Staubli VAL3: StaubliUI.pjx

--- StaubliUI.pjx ---
Parameters version=s7.3.1 stackSize=15000 millimeterUnit=true
Program file=Bool_Edit.pgx
Program file=BoolMess_Edit.pgx
Program file=Control_Action.pgx
Program file=Control_BatPrt.pgx
Program file=Control_BatSpd.pgx
Program file=Control_Bottom.pgx
Program file=Control_BottomS.pgx
Program file=Control_Joint.pgx
Program file=Control_Lable.pgx
Program file=Control_Left.pgx
Program file=Control_LeftS.pgx
Program file=Control_List.pgx
Program file=Control_List1S.pgx
Program file=Control_ListBS.pgx
Program file=Control_ListCls.pgx
Program file=Control_ListMC.pgx
Program file=Control_ListMCD.pgx
Program file=Control_ListMJ.pgx
Program file=Control_ListS.pgx
Program file=Control_Loffset.pgx
Program file=Control_MCShow.pgx
Program file=Control_Mess.pgx
Program file=Control_Panel.pgx
Program file=Control_PanelB.pgx
Program file=Control_PanelD.pgx
Program file=Control_PanelMd.pgx
Program file=Control_PanelS.pgx
Program file=Control_PanelXY.pgx
Program file=Control_Para.pgx
Program file=Control_PatMove.pgx
Program file=Control_Point.pgx
Program file=Control_Preset.pgx
Program file=Control_Recipe.pgx
Program file=Control_Remote.pgx
Program file=Control_Scara.pgx
Program file=Control_Timer.pgx
Program file=Control_Traj.pgx
Program file=Control_YesNO.pgx
Program file=Float_Edit.pgx
Program file=Form_4jHome.pgx
Program file=Form_6jHome.pgx
Program file=Form_Action.pgx
Program file=Form_Bye.pgx
Program file=Form_Config.pgx
Program file=Form_LabelList.pgx
Program file=Form_Main.pgx
Program file=Form_MainS.pgx
Program file=Form_Panel.pgx
Program file=Form_Panel4P.pgx
Program file=Form_PanelBool.pgx
Program file=Form_PanelJoint.pgx
Program file=Form_PanelList.pgx
Program file=Form_PanelPoint.pgx
Program file=Form_PanelStr.pgx
Program file=Form_Patten.pgx
Program file=Form_PattenD.pgx
Program file=Form_PattenS.pgx
Program file=Form_Product.pgx
Program file=Form_ScaraRobot.pgx
Program file=Form_SelSharp.pgx
Program file=Form_Simulation.pgx
Program file=Form_Welcome.pgx
Program file=Int_Edit.pgx
Program file=Int_EditS.pgx
Program file=Key_ListBase.pgx
Program file=Key_ListMC.pgx
Program file=ReadMe.pgx
Program file=Sel_Edit.pgx
Program file=start.pgx
Program file=stop.pgx
Program file=Str_Edit.pgx
Program file=Str_SplitChar.pgx
Program file=Str_SplitComma.pgx
Data file=StaubliUI.dtx

--- start.pgx ---
public program start()
  local num l_nKeyValue
  local bool l_bBool[199]
  local num l_nNum
  local num l_nNum1
  local bool l_brES
begin
  cls()
  //call Control_PanelB("fasdfa","fasdfas")
//  call Frame_PattenD("hELLO")
//  call Control_ListS("1,3,5,6,6,7,8,8,9,90,2,43,5,56",l_nNum)
//  //call Control_YesNO("FDSAFA  AFSDASA",l_brES)
// // call Control_Timer("fasdfafa",5)
////  cls()
////  if l_brES
////    popUpMsg("yes")
////  else
////    popUpMsg("NO")
////  endIf
//   l_bBool[120]=true
//   call Control_ListMC(l_bBool,l_nNum,l_nNum1)
//   call Control_Lable("目前点序号:",l_nNum,0)
//   while true
//
//    call Key_ListMC(l_brES,l_nKeyValue,l_nNum,l_nNum1)
//    if l_brES
//      call Control_ListMC(l_bBool,l_nNum,l_nNum1)
//      call Control_Lable("目前点序号:",l_nNum,0)
//    endIf
//    //使用Q作为快选方式
//    if l_nKeyValue==113
//     call Num_EditS1D(l_nNum,"目前点序号:")
//     call Control_ListMC(l_bBool,l_nNum,l_nNum1)
//     call Control_Lable("目前点序号:",l_nNum,0)
//
//    endIf
//

//
//
//    delay(0)
//  endWhile
//  call Frame_PattenD("hELLO")
   call Control_ListBS("1,2,3,4,5,6","发生大幅，发，发，发，发，发",l_nNum,0)


end

--- Bool_Edit.pgx ---
public program Bool_Edit(bool& x_bRes, num x_nX, num x_nY, num x_nLength)
  local num l_nNum
  local string l_s[2]
begin

  l_s[1]="是"
  l_s[0]="否"


   call BoolMess_Edit(x_bRes,x_nX,x_nY,x_nLength,l_s)

end

--- BoolMess_Edit.pgx ---
public program BoolMess_Edit(bool& x_bRes, num x_nX, num x_nY, num x_nLength, string& x_sMess[])
  local num l_nNum
begin


   l_nNum=sel(x_bRes,1,0)
   call Sel_Edit(l_nNum,x_nX,x_nY,x_sMess)
   x_bRes=(l_nNum==1)

end

--- Control_Action.pgx ---
public program Control_Action(num& x_nAction[] (dimensions=3), num x_nIndex, string& x_sIoName[], bool& x_bDigtal[])
  local string l_sItem[2]
  local num l_nNum
  local num l_nKey
  local num l_nData[24]
  local num l_nSelectIndex
  local bool l_bRes
begin

  //修改点位的 joint

  for l_nNum=0 to 11
    l_nData[l_nNum*2+0]=x_nAction[x_nIndex,l_nNum,0]
    l_nData[l_nNum*2+1]=x_nAction[x_nIndex,l_nNum,1]
  endFor
  l_sItem[0]="关"
  l_sItem[1]="开"

  resize(sBuff,1,24)


  call Control_BottomS("置空,清空,延时,,,,取消,确定")
  call Control_PanelXY(4,0,20,10)
  call Control_Panel("动作值")
  for l_nNum=0 to 11


    sBuff[l_nNum*2+0]=toString("",l_nNum+1)+"名称:"+x_sIoName[l_nData[l_nNum*2+0]]
    if x_bDigtal[l_nData[l_nNum*2]]
      sBuff[l_nNum*2+1]="值 : "+ l_sItem[sel(l_nData[l_nNum*2+1]==0,0,1)]
    else
      sBuff[l_nNum*2+1]="值 : "+toString("",l_nData[l_nNum*2+1])
    endIf

  endFor
  call Control_List(sBuff,l_nSelectIndex)


  //**********************************
  //按键响应
  while true
    l_nKey=getKey()

    switch l_nKey
      //向上
      case 261
        l_nSelectIndex=max(0,l_nSelectIndex-1)
      break

      //向下
      case 266
        l_nSelectIndex=min(l_nSelectIndex+1,23)
      break

      //编辑
      case 270
        if l_nSelectIndex%2==1
          if ! x_bDigtal[l_nData[l_nSelectIndex-1]]
            call Float_Edit(l_nData[l_nSelectIndex],nPanelLTopX+6,l_nSelectIndex+nPanelLTopY+1)
          else
            call Sel_Edit(l_nData[l_nSelectIndex],nPanelLTopX+6,l_nSelectIndex+nPanelLTopY+1,l_sItem)
          endIf

        else
          call Sel_Edit(l_nData[l_nSelectIndex],nPanelLTopX+7,l_nSelectIndex+nPanelLTopY+1,x_sIoName)
        endIf

      break

      case 271
        call Control_YesNO("确定设置为无IO信号吗?",l_bRes)
        if l_bRes

          l_nData[sel(l_nSelectIndex%2==0,l_nSelectIndex,l_nSelectIndex-1)]=0

        endIf

      break


      //全部置空
      case 272
        call Control_YesNO("确定全部清空吗?",l_bRes)
        if l_bRes
          for l_nNum=0 to 23
            l_nData[l_nNum]=0
          endFor


        endIf
      break


      case 273
        call Control_YesNO("确定要设置为延时吗?",l_bRes)
        if l_bRes
          l_nData[sel(l_nSelectIndex%2==0,l_nSelectIndex,l_nSelectIndex-1)]=165

        endIf
      break


      //退出
      case 277
        cls()
        return

      break



      //取消
      case 278
        for l_nNum=0 to 11
          x_nAction[x_nIndex,l_nNum,0]= l_nData[l_nNum*2+0]
          x_nAction[x_nIndex,l_nNum,1]=l_nData[l_nNum*2+1]
        endFor
        return
      break

    endSwitch

    if l_nKey!=-1

      for l_nNum=0 to 11
        sBuff[l_nNum*2+0]=toString("",l_nNum+1)+"名称:"+x_sIoName[l_nData[l_nNum*2+0]]
        if x_bDigtal[l_nData[l_nNum*2]]
          sBuff[l_nNum*2+1]="值 : "+ l_sItem[sel(l_nData[l_nNum*2+1]==0,0,1)]
        else
          sBuff[l_nNum*2+1]="值 : "+toString("",l_nData[l_nNum*2+1])
        endIf

      endFor

      call Control_PanelXY(4,0,20,10)
      call Control_Panel("动作值")
      call Control_List(sBuff,l_nSelectIndex)
      call Control_BottomS("置空,清空,延时,,,,取消,确定")
    endIf


  endWhile





end

--- Control_BatPrt.pgx ---
public program Control_BatPrt(num& x_nFrom, num& x_nTo, num& x_nPreset)
  local string l_sItem[3]
  local num l_nNum
  local num l_nKey
  local num l_nData[6]
  local num l_nSelectIndex
begin

  //修改点位的 joint
  l_nData[0]=x_nFrom
  l_nData[1]=x_nTo
  l_nData[2]=1
  //l_nData[3]=15
  l_sItem[0]="开始    :"+toString("",l_nData[0])
  l_sItem[1]="结束    :"+toString("",l_nData[1])
  l_sItem[2]="工艺    :"+toString("",l_nData[2])
  //  l_sItem[3]="加速度  :"+toString("",l_nData[3])



  call Control_BottomS(",,,,,,取消,确定")
  call Control_PanelXY(8,0,15,4)
  call Control_Panel("批处理工艺")
  call Control_List(l_sItem,l_nSelectIndex)
  while true
    l_nKey=getKey()

    switch l_nKey
      case 261
        l_nSelectIndex=max(0,l_nSelectIndex-1)
      break

      case 266
        l_nSelectIndex=min(l_nSelectIndex+1,2)
      break

      case 278
        x_nFrom=l_nData[0]
        x_nTo=l_nData[1]
        x_nPreset=l_nData[2]
        //   x_nAcc=l_nData[3]
        cls()
        return
      break


      case 277,255

        cls()
        return
      break

      case 270
        call Float_Edit(l_nData[l_nSelectIndex],nPanelLTopX+7,l_nSelectIndex+nPanelLTopY+1)
      break

    endSwitch

    if l_nKey!=-1
      l_nData[2]=min(max(1,l_nData[2]),50)
      l_nData[2]=round(l_nData[2])
      l_sItem[0]="开始    :"+toString("",l_nData[0])
      l_sItem[1]="结束    :"+toString("",l_nData[1])
      l_sItem[2]="工艺    :"+toString("",l_nData[2])
      // l_sItem[3]="加速度  :"+toString("",l_nData[3])
      call Control_List(l_sItem,l_nSelectIndex)

    endIf






  endWhile





end

--- Control_BatSpd.pgx ---
public program Control_BatSpd(num& x_nFrom, num& x_nTo, num& x_nSpeed, num& x_nAcc)
  local string l_sItem[4]
  local num l_nNum
  local num l_nKey
  local num l_nData[6]
  local num l_nSelectIndex
begin

  //修改点位的 joint
  l_nData[0]=x_nFrom
  l_nData[1]=x_nTo
  l_nData[2]=100
  l_nData[3]=15
  l_sItem[0]="开始    :"+toString("",l_nData[0])
  l_sItem[1]="结束    :"+toString("",l_nData[1])
  l_sItem[2]="速度    :"+toString("",l_nData[2])
  l_sItem[3]="加速度  :"+toString("",l_nData[3])



  call Control_BottomS(",,,,,,取消,确定")
  call Control_PanelXY(8,0,15,4)
  call Control_Panel("批处理速度")
  call Control_List(l_sItem,l_nSelectIndex)
  while true
    l_nKey=getKey()

    switch l_nKey
      case 261
        l_nSelectIndex=max(0,l_nSelectIndex-1)
      break

      case 266
        l_nSelectIndex=min(l_nSelectIndex+1,3)
      break

      case 278
        x_nFrom=l_nData[0]
        x_nTo=l_nData[1]
        x_nSpeed=l_nData[2]
        x_nAcc=l_nData[3]
        cls()
        return
      break


      case 277,255

        cls()
        return
      break

      case 270
        call Float_Edit(l_nData[l_nSelectIndex],nPanelLTopX+7,l_nSelectIndex+nPanelLTopY+1)
      break

    endSwitch

    if l_nKey!=-1
  l_sItem[0]="开始    :"+toString("",l_nData[0])
  l_sItem[1]="结束    :"+toString("",l_nData[1])
  l_sItem[2]="速度    :"+toString("",l_nData[2])
  l_sItem[3]="加速度  :"+toString("",l_nData[3])
      call Control_List(l_sItem,l_nSelectIndex)

    endIf






  endWhile





end

--- Control_Bottom.pgx ---
public program Control_Bottom(string& x_sBottomList[])
  local num l_nIndex
  local num l_nNum
begin
  //说明：
  //函数功能：对功能键进行说明
  //


  //参数初始化
  setTextMode(0)
  l_nNum=min(7,size(x_sBottomList)-1)


  for l_nIndex=0 to  l_nNum
    gotoxy(1+l_nIndex*5,13)
    put(left(x_sBottomList[l_nIndex]+"       ",4+len(x_sBottomList[l_nIndex])-getDisplayLen(x_sBottomList[l_nIndex])))
  endFor

  //补全
  if l_nNum<7
    for l_nIndex=l_nNum to 7
      gotoxy(1+l_nIndex*5,13)
      put("  ")
    endFor
  endIf
end

--- Control_BottomS.pgx ---
public program Control_BottomS(string x_sBottomList)
  local string l_sBottomList[8]
  local bool l_bRes
begin

  call Str_SplitComma(l_bRes,x_sBottomList,l_sBottomList)
  if !l_bRes
    return
  endIf

call Control_Bottom(l_sBottomList)

end

--- Control_Joint.pgx ---
public program Control_Joint(jointRx& x_jJ)
  local string l_sItem[6]
  local num l_nNum
  local num l_nKey
  local num l_nData[6]
  local num l_nSelectIndex
begin

  //修改点位的 joint
  l_nData[0]=x_jJ.j1
  l_nData[1]=x_jJ.j2
  l_nData[2]=x_jJ.j3
  l_nData[3]=x_jJ.j4
  l_nData[4]=x_jJ.j5
  l_nData[5]=x_jJ.j6

  for l_nNum=0 to 5
    l_sItem[l_nNum]="j"+toString("",l_nNum+1)+"   :"+toString(".3",l_nData[l_nNum])
  endFor

  call Control_BottomS(",,,,,,取消,确定")
  call Control_PanelXY(8,0,15,6)
  call Control_Panel("Joint值")
  call Control_List(l_sItem,l_nSelectIndex)
  while true
    l_nKey=getKey()

    switch l_nKey
      case 261
        l_nSelectIndex=max(0,l_nSelectIndex-1)
      break

      case 266
        l_nSelectIndex=min(l_nSelectIndex+1,5)
      break

      case 278
        x_jJ.j1=l_nData[0]
        x_jJ.j2=l_nData[1]
        x_jJ.j3=l_nData[2]
        x_jJ.j4=l_nData[3]
        x_jJ.j5=l_nData[4]
        x_jJ.j6=l_nData[5]
        return
      break


      case 277,255
        return
      break

      case 270
        call Float_Edit(l_nData[l_nSelectIndex],nPanelLTopX+7,l_nSelectIndex+nPanelLTopY+1)
      break

    endSwitch

    if l_nKey!=-1
      for l_nNum=0 to 5
        l_sItem[l_nNum]="j"+toString("",l_nNum+1)+"   :"+toString(".3",l_nData[l_nNum])
      endFor
      call Control_List(l_sItem,l_nSelectIndex)

    endIf






  endWhile





end

--- Control_Lable.pgx ---
public program Control_Lable(string x_sMess, num& Value, num x_nTextMode)
begin
setTextMode(0)
gotoxy(0,0)
put(x_sMess)
gotoxy(getDisplayLen(x_sMess),0)
x_nTextMode=min(max(0,x_nTextMode),3)
setTextMode(x_nTextMode)
//序号加1
put(left(toString("",Value+1)+"            ",max(8,nPanelLTopX-getDisplayLen(x_sMess)-len(toString("",Value)))))
setTextMode(0)
end

--- Control_Left.pgx ---
program Control_Left(string& x_sLeftList[])
  local num l_nIndex
begin

    setTextMode(0)
  //左边栏进行显示
  for l_nIndex=0 to min(7,size(x_sLeftList)-1)
    gotoxy(1,l_nIndex+4)
    if size(x_sLeftList)>l_nIndex and x_sLeftList[l_nIndex]!=""
      put("F"+toString("",l_nIndex+1)+"->"+x_sLeftList[l_nIndex])
    endIf
  endFor
end

--- Control_LeftS.pgx ---
public program Control_LeftS(string x_sLeftList)
  local bool l_bRes
  local string l_sBuff[20]
begin

  call Str_SplitComma(l_bRes,x_sLeftList,l_sBuff)
  if !l_bRes
    return
  endIf

call Control_Left(l_sBuff)
end

--- Control_List.pgx ---
public program Control_List(string& x_sItemName[], num& x_nSelectItem)
  local num l_nIndex
  local bool l_bRes
  local num l_nFrist
  local num l_nNum
  local bool l_bBlack
  local bool l_bBlank
  local num l_nCount
begin
  //说明：
  //函数功能：在划定的框内，把选中项给显示出来
  //l_nFirst  在列表中第一个显示的项的序号
  //x_nSelectItem  被选中的项的序号
  //l_nCount 合法列表项的项总数，如何数组中间为空，则可能被截断


  //1.参数初始化
  l_nFrist=0
  l_nCount=0

  //2.参数合法化判断，得到合法项的总数
  for l_nIndex=0 to size(x_sItemName)-1
    if x_sItemName[l_nIndex]==""
      l_nIndex=size(x_sItemName)
    else
      l_nCount=l_nCount+1
    endIf
  endFor

  //3.如果选中项大于列表长度
  x_nSelectItem=min(max(0,x_nSelectItem),l_nCount-1)
  if x_nSelectItem>=nPanelLengthY
    l_nFrist=x_nSelectItem-nPanelLengthY+1
  endIf


  //4.把列表给画出来
  for l_nIndex=0 to min(nPanelLengthY-1,l_nCount-l_nFrist-1)
    gotoxy(nPanelLTopX+1,nPanelLTopY+l_nIndex+1)
    setTextMode(sel(l_nIndex+l_nFrist==x_nSelectItem,1,0))
    l_nNum=nPanelWidthX-getDisplayLen(x_sItemName[l_nIndex+l_nFrist])+len(x_sItemName[l_nIndex+l_nFrist])
    put(left(x_sItemName[l_nIndex+l_nFrist]+"                            ",l_nNum))
  endFor


  //5.对剩下的进行补空
  setTextMode(0)
  while l_nIndex< nPanelLengthY
    gotoxy(nPanelLTopX+1,nPanelLTopY+l_nIndex+1)
    put(left("                               ",nPanelWidthX-2))
    l_nIndex=l_nIndex+1
  endWhile


end

--- Control_List1S.pgx ---
public program Control_List1S(string x_sItemName, string x_sItemValue, num x_nSelectItem, num x_nText)
  local string l_sBuff[10]
  local string l_sValue[10]
  local num l_nIndex
  local bool l_bRes
begin
   // 赋初值
   for l_nIndex=0 to size(l_sBuff)-1
    l_sBuff[l_nIndex]=""
  endFor

  //把项的名字给解析出来
  call  Str_SplitChar(l_bRes,x_sItemName,",",l_sBuff)
  if !l_bRes
    return
  endIf

    call  Str_SplitChar(l_bRes,x_sItemValue,",",l_sValue)
  if !l_bRes
    return
  endIf


  //对方框的定义进行赋初值
  // call Control_ListBas(x_nSelectItem)


  //把列表给画出来
  for l_nIndex=0 to min(min(nPanelLengthY-1,size(l_sBuff)-1),size(l_sValue)-1)
    if l_sBuff[l_nIndex]==""
      return
    endIf
    setTextMode(0)
    gotoxy(nPanelLTopX+1,nPanelLTopX+l_nIndex+1)
    put(left(l_sBuff[l_nIndex]+"              ",nPanelWidthX-getDisplayLen(l_sBuff[l_nIndex])+len(l_sBuff[l_nIndex]))+":")
    gotoxy(nPanelLTopX+nPanelWidthX/2-getDisplayLen(l_sBuff[l_nIndex])+len(l_sBuff[l_nIndex]),nPanelLTopY+l_nIndex+1)
    //选中项变成黑色
    if l_nIndex==x_nSelectItem

      setTextMode(x_nText)
    endIf

    //直接截取+
    //中文编码与英文编码有点不一样
    put(left(l_sValue[l_nIndex]+"             ",nPanelWidthX/2-getDisplayLen(l_sValue[l_nIndex])+len(l_sValue[l_nIndex])))

  endFor


end

--- Control_ListBS.pgx ---
public program Control_ListBS(string x_sItemName, string x_sItemValue, num x_nSelectItem, num x_nText)
  local string l_sBuff[10]
  local string l_sValue[10]
  local num l_nIndex
  local bool l_bRes
begin
   // 赋初值
   for l_nIndex=0 to size(l_sBuff)-1
    l_sBuff[l_nIndex]=""
  endFor

  //把项的名字给解析出来
  call  Str_SplitComma(l_bRes,x_sItemName,l_sBuff)
  if !l_bRes
    return
  endIf

    call  Str_SplitComma(l_bRes,x_sItemValue,l_sValue)
  if !l_bRes
    return
  endIf

  call Control_PanelXY(nPanelLTopX,nPanelLTopY,nPanelWidthX/2,nPanelLengthY)
  call Control_List(l_sBuff,x_nSelectItem)
  call Control_PanelXY(nPanelLTopX+nPanelWidthX/2,nPanelLTopY,nPanelWidthX/2,nPanelLengthY)
  call Control_List(l_sValue,x_nSelectItem)

end

--- Control_ListCls.pgx ---
program Control_ListCls()
  local num l_nIndex
begin



  //对方框的定义进行赋初值
  if nPanelLengthY<=0 and nPanelLTopX<=0 and nPanelLTopY<=0 and nPanelWidthX<=0
    call Control_PanelXY(20,0,18,11)
  endIf

  //清空列表
  setTextMode(0)
  for l_nIndex=0 to nPanelLengthY-1
    gotoxy(nPanelLTopX+1,nPanelLTopY+l_nIndex+1)
    put(left("                                               ",nPanelWidthX))
  endFor

  //参数判断  对于选择项的判断
 // x_nSelectItem=min(max(0,x_nSelectItem),nPanelLengthY-1)


end

--- Control_ListMC.pgx ---
public program Control_ListMC(bool& x_bMC[], num& x_nSelectItem, num x_nText)
  local num l_nIndex
  local bool l_bRes
  local string l_sText
  local num l_nFrist
begin
   //赋初值
   // call Control_ListCls()

    l_nFrist=0
  x_nSelectItem=min(max(0,x_nSelectItem),size(x_bMC)-1)
  if x_nSelectItem>=nPanelLengthY
    l_nFrist=x_nSelectItem-nPanelLengthY+1
  endIf


  //把列表给画出来
  for l_nIndex=0 to min(nPanelLengthY-1,size(x_bMC)-l_nFrist)
    gotoxy(nPanelLTopX+1,nPanelLTopY+l_nIndex+1)
    //选中项变成黑色


    //MOVEL
    if !x_bMC[l_nIndex+l_nFrist]
      if l_nIndex+l_nFrist==x_nSelectItem

        setTextMode(1)
      else
        setTextMode(0)
      endIf
      put(left(toString("",l_nIndex+l_nFrist+1)+"       ",5 )+left("MOVEL             ",nPanelWidthX-5))
    else

    //MOVEC
       setTextMode(0)
      put(left("                                               ",nPanelWidthX))
      gotoxy(nPanelLTopX+1,nPanelLTopY+l_nIndex+1)
      if l_nIndex+l_nFrist!=x_nSelectItem
        put(left(toString("",l_nIndex+l_nFrist+1)+"       ",5 )+left("MOVEC Pc Pt              ",nPanelWidthX-5))
      else
        if x_nText==0
          setTextMode(1)
        else
          setTextMode(0)
        endIf
        put(left(toString("",l_nIndex+l_nFrist+1)+"       ",5 )+"MOVEC")
        gotoxy(nPanelLTopX+12,nPanelLTopY+l_nIndex+1)
        if x_nText==1

          setTextMode(1)
        else
          setTextMode(0)
        endIf
        put("Pc")
        //目标点
        gotoxy(nPanelLTopX+15,nPanelLTopY+l_nIndex+1)

        if x_nText==2
          setTextMode(1)
        else
          setTextMode(0)
        endIf
        put("Pt")
      endIf
    endIf
  endFor

   setTextMode(0)
  while l_nIndex< nPanelLengthY
    gotoxy(nPanelLTopX+1,nPanelLTopY+l_nIndex+1)
    put(left("                          ",nPanelWidthX-2))
    l_nIndex=l_nIndex+1
  endWhile

end

--- Control_ListMCD.pgx ---
public program Control_ListMCD(bool& x_bMC[], num& x_nSelectItem, num& x_nText)
  local num l_nIndex
  local bool l_bRes
  local string l_sText
  local num l_nFrist
begin
   //赋初值
   // call Control_ListCls()

    l_nFrist=0
  x_nSelectItem=min(max(0,x_nSelectItem),size(x_bMC)-1)
  if x_nSelectItem>=nPanelLengthY
    l_nFrist=x_nSelectItem-nPanelLengthY+1
  endIf


  //把列表给画出来
  for l_nIndex=0 to min(nPanelLengthY-1,size(x_bMC)-l_nFrist)
    gotoxy(nPanelLTopX+1,nPanelLTopY+l_nIndex+1)
    //选中项变成黑色


    //MOVEL
    if !x_bMC[l_nIndex+l_nFrist]
      if l_nIndex+l_nFrist==x_nSelectItem
          if x_nText==0
          setTextMode(1)
        else
          setTextMode(0)
        endIf
        put(left(toString("",l_nIndex+l_nFrist+1)+"       ",5 )+"MOVEL")
        gotoxy(nPanelLTopX+12,nPanelLTopY+l_nIndex+1)
        if x_nText==1

          setTextMode(1)
        else
          setTextMode(0)
        endIf
        put("Pl")
      else
        setTextMode(0)
        put(left(toString("",l_nIndex+l_nFrist+1)+"       ",5 )+left("MOVEL Pl             ",nPanelWidthX-5))
      endIf

    else

    //MOVEC
       setTextMode(0)
      put(left("                                               ",nPanelWidthX))
      gotoxy(nPanelLTopX+1,nPanelLTopY+l_nIndex+1)
      if l_nIndex+l_nFrist!=x_nSelectItem
        put(left(toString("",l_nIndex+l_nFrist+1)+"       ",5 )+left("MOVEC Pc Pt              ",nPanelWidthX-5))
      else
        if x_nText==0
          setTextMode(1)
        else
          setTextMode(0)
        endIf
        put(left(toString("",l_nIndex+l_nFrist+1)+"       ",5 )+"MOVEC")
        gotoxy(nPanelLTopX+12,nPanelLTopY+l_nIndex+1)
        if x_nText==1

          setTextMode(1)
        else
          setTextMode(0)
        endIf
        put("Pc")
        //目标点
        gotoxy(nPanelLTopX+15,nPanelLTopY+l_nIndex+1)

        if x_nText==2
          setTextMode(1)
        else
          setTextMode(0)
        endIf
        put("Pt")
      endIf
    endIf
  endFor

   setTextMode(0)
  while l_nIndex< nPanelLengthY
    gotoxy(nPanelLTopX+1,nPanelLTopY+l_nIndex+1)
    put(left("                          ",nPanelWidthX-2))
    l_nIndex=l_nIndex+1
  endWhile

end

--- Control_ListMJ.pgx ---
public program Control_ListMJ(bool& x_bMJ[], num x_nMoveFirst, num x_nSelectItem)
  local num l_nIndex
  local bool l_bRes
  local string l_sText
begin


//  call Control_ListBas(x_nSelectItem)
//
//
//
//
//  //把列表给画出来
//  for l_nIndex=0 to min(nBottomY-nTopY-1,size(x_bMJ)-x_nMoveFirst)
//
//    setTextMode(0)
//    if x_nMoveFirst+l_nIndex>size(x_bMJ)-1
//      return
//    endIf
//    //MOVEL
//    gotoxy(nTopX+1,nTopY+l_nIndex+1)
//    if !x_bMJ[x_nMoveFirst+l_nIndex]
//      if l_nIndex==x_nSelectItem
//        setTextMode(1)
//      else
//        setTextMode(0)
//      endIf
//      put(left(toString("",x_nMoveFirst+l_nIndex+1)+"       ",4 )+left("MOVEJ             ",24-nBottomX))
//    else
//      //MOVEC
//      if l_nIndex==x_nSelectItem
//        setTextMode(1)
//      else
//        setTextMode(0)
//      endIf
//      put(left(toString("",x_nMoveFirst+l_nIndex+1)+"       ",4 )+left("MOVEL              ",24-nBottomX))
//
//    endIf
//
//  endFor
//

end

--- Control_ListS.pgx ---
program Control_ListS(string x_sItemName, num& x_nSelectItem)
  local bool l_bRes
  local string l_sBuff[20]
begin

 call Str_SplitComma(l_bRes,x_sItemName,l_sBuff)
 if !l_bRes
  return
endIf
  call Control_List(l_sBuff,x_nSelectItem)


end

--- Control_Loffset.pgx ---
public program Control_Loffset(num& x_nFrom, num& x_nTo)
  local string l_sItem[2]
  local num l_nNum
  local num l_nKey
  local num l_nData[6]
  local num l_nSelectIndex
begin

  //修改点位的 joint
l_nData[0]=x_nFrom
l_nData[1]=x_nTo

  l_sItem[0]="开始    :"+toString("",l_nData[0])
  l_sItem[1]="停止    :"+toString("",l_nData[1])
  call Control_BottomS(",,,,,,取消,确定")
  call Control_PanelXY(8,0,15,6)
  call Control_Panel("局部偏差值")
  call Control_List(l_sItem,l_nSelectIndex)
  while true
    l_nKey=getKey()

    switch l_nKey
      case 261
        l_nSelectIndex=max(0,l_nSelectIndex-1)
      break

      case 266
        l_nSelectIndex=min(l_nSelectIndex+1,1)
      break

      case 278
          x_nFrom=l_nData[0]
          x_nTo=l_nData[1]
         cls()
        return
      break


      case 277,255

        cls()
        return
      break

      case 270
        call Float_Edit(l_nData[l_nSelectIndex],nPanelLTopX+7,l_nSelectIndex+nPanelLTopY+1)
      break

    endSwitch

    if l_nKey!=-1
  l_sItem[0]="开始    :"+toString("",l_nData[0])
  l_sItem[1]="停止    :"+toString("",l_nData[1])
      call Control_List(l_sItem,l_nSelectIndex)

    endIf






  endWhile





end

--- Control_MCShow.pgx ---
public program Control_MCShow(num x_nIndex, num x_nMoveType)
  local string l_sS[3]
begin
  if x_nMoveType>2 or x_nMoveType<1
    return
  endIf
  l_sS[0]=toString("",x_nIndex+1)+"."+"MoveC "
  l_sS[1]=toString("",1)+" "
  l_sS[2]=left(" "+toString("",2)+"       ",nPanelWidthX-len(l_sS[0])-len(l_sS[1]))
  setTextMode(0)
  gotoxy(nPanelLTopX+1,min(nPanelLengthY,x_nIndex+1))
  put(l_sS[0])
  setTextMode(sel(x_nMoveType==1,1,0))
  put(l_sS[1])
  setTextMode(sel(x_nMoveType==1,0,1))
  put(l_sS[2])


  setTextMode(0)

end

--- Control_Mess.pgx ---
public program Control_Mess(string x_sMess, string x_sLable)
begin

  setTextMode(0)
gotoxy(0,1)
put(x_sMess)
  gotoxy(0,2)
put(x_sLable)

end

--- Control_Panel.pgx ---
program Control_Panel(string x_sTitle)
  local num l_nIndex
  local string l_sS
begin
  //画框函数
  //如果标题为空，



    setTextMode(0)

  //方框进行重画

  //画上边
   gotoxy(nPanelLTopX,nPanelLTopY)
   l_sS="┌"+left("───────────────────────────────────",nPanelWidthX)

  //写标题

     //2是两个标志符
  if x_sTitle!=""
    x_sTitle=left(x_sTitle,min(getDisplayLen(x_sTitle),nPanelWidthX)-getDisplayLen(x_sTitle)+len(x_sTitle))
    x_sTitle="┤"+x_sTitle+"├┐"
    l_sS=left(l_sS,nPanelWidthX-getDisplayLen(x_sTitle)+2)+x_sTitle
  else
    l_sS=l_sS+"┐"
  endIf
  put(l_sS)

   //画下边
   gotoxy(nPanelLTopX,nPanelLTopY+nPanelLengthY+1)
   put("└"+left("─────────────────────────────────────────",nPanelWidthX)+"┘")

   //重画两边
   for l_nIndex=1 to nPanelLengthY
    gotoxy(nPanelLTopX,nPanelLTopY+l_nIndex)
   // put("│")
   put("│")
    gotoxy(nPanelLTopX+nPanelWidthX+1,nPanelLTopY+l_nIndex)
    put("│")
  endFor












end

--- Control_PanelB.pgx ---
public program Control_PanelB(string x_sLeftTitle, string x_sRightTitle)
begin
    //两个方框
   call Control_PanelS(x_sLeftTitle,0,0,18,11)

   call Control_PanelS(x_sRightTitle,20,0,18,11)

end

--- Control_PanelD.pgx ---
public program Control_PanelD()
begin
  call Control_PanelS("",20,0,18,11)


end

--- Control_PanelMd.pgx ---
public program Control_PanelMd(string x_sMess)
begin

  call Control_PanelS("",2,3,34,4)
  call Control_ListCls()
  x_sMess=left(x_sMess,min(getDisplayLen(x_sMess),nPanelWidthX))
  gotoxy(nPanelLTopX+ (nPanelWidthX-getDisplayLen(x_sMess))/2,nPanelLTopY+nPanelLengthY/2+1)
  put( x_sMess)


end

--- Control_PanelS.pgx ---
public program Control_PanelS(string x_sTitle, num x_nLTopX, num x_nLTopY, num x_nWidthX, num x_nLengthY)
  local num l_nIndex
begin
  //画有标题的框



  //设定框的位置与大小
  call Control_PanelXY(x_nLTopX,x_nLTopY,x_nWidthX,x_nLengthY)

  //文本显示状况进行设定
   call Control_Panel(x_sTitle)









end

--- Control_PanelXY.pgx ---
public program Control_PanelXY(num x_nPanelLTopX, num x_nPanelLTopY, num x_nPanelWidthX, num x_nPanelLengthY)
begin

//对于新建的框和列表进行位置和大小的设定

//对于数值范围进行判断，一般的情况可以使用min,max就可以
//如果传入的参数不正确，则设定初始值
nPanelLTopX=min(max(0,x_nPanelLTopX),38)
nPanelLTopY=min(max(0,x_nPanelLTopY),12)

nPanelWidthX=min(max(0,x_nPanelWidthX),38)
nPanelLengthY=min(max(0,x_nPanelLengthY),12)


end

--- Control_Para.pgx ---
public program Control_Para(trsf& x_trTrsf, bool& x_bRes, bool x_bCut, num x_nType)
  local string l_sItem[6]
  local num l_nNum
  local num l_nKey
  local num l_nData[6]
  local num l_nSelectIndex
begin

  //修改点位的 joint
  l_nData[3]=x_trTrsf.x
  l_nData[4]=x_trTrsf.y
  l_nData[0]=x_trTrsf.z
  l_nData[1]=x_trTrsf.rx

  l_nData[2]=x_trTrsf.ry
  l_nData[5]=x_trTrsf.rz
  l_nNum=sel(x_bRes,1,0)
  resize(sData,1,2)
  if x_bCut

    sData[0]="直线"
    sData[1]="圆弧"
    l_sItem[0]="速度(mm/s:"+toString(".3",l_nData[0])
    l_sItem[1]="加速度(%):"+toString(".3",l_nData[1])
    l_sItem[2]="BLend(mm):"+toString(".3",l_nData[2])
    l_sItem[3]="工艺     :"+toString(".3",l_nData[3])
    l_sItem[4]="动作     :"+toString(".3",l_nData[4])
    l_sItem[5]="圆弧/直线:"+sData[l_nNum]

  else
    sData[0]="MoveJ"
    sData[1]="MoveL"
    l_sItem[0]="速度(mm/s:"+toString(".3",l_nData[0])
    l_sItem[1]="加速度(%):"+toString(".3",l_nData[1])
    l_sItem[2]="关节/直线:"+sData[l_nNum]

  endIf

  call Control_BottomS(",,,,,,取消,确定")
  if x_bCut
    if x_nType!=10
      call Control_PanelXY(8,0,18,5)
    else
      call Control_PanelXY(8,0,18,6)
    endIf
  else
    call Control_PanelXY(8,0,17,3)
  endIf
  call Control_Panel("参数")
  call Control_List(l_sItem,l_nSelectIndex)
  while true
    l_nKey=getKey()

    switch l_nKey
      case 261
        l_nSelectIndex=max(0,l_nSelectIndex-1)
      break

      case 266
        if x_bCut
          if x_nType==10
            l_nSelectIndex=min(l_nSelectIndex+1,5)
          else
            l_nSelectIndex=min(l_nSelectIndex+1,4)
          endIf
        else
          l_nSelectIndex=min(l_nSelectIndex+1,2)
        endIf
      break

      case 278
        x_trTrsf.x=l_nData[3]
        x_trTrsf.y=l_nData[4]
        x_trTrsf.z=l_nData[0]
        x_trTrsf.rx=l_nData[1]

        x_trTrsf.ry=l_nData[2]
        x_trTrsf.rz=l_nData[5]
        x_bRes=(l_nNum==1)
        cls()
        return
      break


      case 277,255
        cls()
        return
      break



      case 270
        if (l_nSelectIndex==2 and !x_bCut) or (l_nSelectIndex==5 and x_bCut)
          call Sel_Edit(l_nNum,nPanelLTopX+11,l_nSelectIndex+nPanelLTopY+1,sData)

        else
          call Float_Edit(l_nData[l_nSelectIndex],nPanelLTopX+11,l_nSelectIndex+nPanelLTopY+1)
        endIf
      break

    endSwitch

    if l_nKey!=-1
      if x_bCut

        sData[0]="直线"
        sData[1]="圆弧"
        l_sItem[0]="速度(mm/s:"+toString(".3",l_nData[0])
        l_sItem[1]="加速度(%):"+toString(".3",l_nData[1])
        l_sItem[2]="BLend(mm):"+toString(".3",l_nData[2])
        l_sItem[3]="工艺     :"+toString(".3",l_nData[3])
        l_sItem[4]="动作     :"+toString(".3",l_nData[4])
        l_sItem[5]="圆弧/直线:"+sData[l_nNum]

      else
        sData[0]="MoveJ"
        sData[1]="MoveL"
        l_sItem[0]="速度(mm/s:"+toString(".3",l_nData[0])
        l_sItem[1]="加速度(%):"+toString(".3",l_nData[1])
        l_sItem[2]="关节/直线:"+sData[l_nNum]

      endIf
      call Control_List(l_sItem,l_nSelectIndex)

    endIf






  endWhile





end

--- Control_PatMove.pgx ---
public program Control_PatMove(num& x_nStart, num& x_nEnd)
  local string l_sItem[6]
  local num l_nNum
  local num l_nKey
  local num l_nData[6]
  local num l_nSelectIndex
begin

  //修改点位的 joint
  l_nData[0]=x_nStart
  l_nData[1]=x_nEnd


  l_sItem[0]="开始模拟点:"+toString(".3",l_nData[0])
  l_sItem[1]="结束模拟点:"+toString(".3",l_nData[1])


  call Control_BottomS(",,,,,,,确定")
  call Control_PanelXY(8,0,15,2)
  call Control_Panel("切割点局部模拟")
  call Control_List(l_sItem,l_nSelectIndex)
  while true
    l_nKey=getKey()

    switch l_nKey
      case 261
        l_nSelectIndex=max(0,l_nSelectIndex-1)
      break

      case 266
        l_nSelectIndex=min(l_nSelectIndex+1,1)
      break

      case 278
        x_nStart=l_nData[0]
        x_nEnd=l_nData[1]
         cls()
        return
      break


//      case 277,255
//
//        cls()
//        return
//      break

      case 270
        call Float_Edit(l_nData[l_nSelectIndex],nPanelLTopX+12,l_nSelectIndex+nPanelLTopY+1)
      break

    endSwitch

    if l_nKey!=-1
  l_sItem[0]="开始模拟点:"+toString(".3",l_nData[0])
  l_sItem[1]="结束模拟点:"+toString(".3",l_nData[1])

      call Control_List(l_sItem,l_nSelectIndex)

    endIf






  endWhile





end

--- Control_Point.pgx ---
public program Control_Point(pointRx& x_pP)
  local string l_sItem[6]
  local num l_nNum
  local num l_nKey
  local num l_nData[6]
  local num l_nSelectIndex
begin

  //修改点位的 joint
  l_nData[0]=x_pP.trsf.x
  l_nData[1]=x_pP.trsf.y
  l_nData[2]=x_pP.trsf.z
  l_nData[3]=x_pP.trsf.rx
  l_nData[4]=x_pP.trsf.ry
  l_nData[5]=x_pP.trsf.rz

  l_sItem[0]="X    :"+toString(".3",l_nData[0])
  l_sItem[1]="y    :"+toString(".3",l_nData[1])
  l_sItem[2]="Z    :"+toString(".3",l_nData[2])
  l_sItem[3]="RX   :"+toString(".3",l_nData[3])
  l_sItem[4]="RY   :"+toString(".3",l_nData[4])
  l_sItem[5]="RZ   :"+toString(".3",l_nData[5])

  call Control_BottomS(",,,,,,取消,确定")
  call Control_PanelXY(8,0,15,6)
  call Control_Panel("Point值")
  call Control_List(l_sItem,l_nSelectIndex)
  while true
    l_nKey=getKey()

    switch l_nKey
      case 261
        l_nSelectIndex=max(0,l_nSelectIndex-1)
      break

      case 266
        l_nSelectIndex=min(l_nSelectIndex+1,5)
      break

      case 278
        x_pP.trsf.x=l_nData[0]
        x_pP.trsf.y=l_nData[1]
        x_pP.trsf.z=l_nData[2]
        x_pP.trsf.rx=l_nData[3]
        x_pP.trsf.ry=l_nData[4]
        x_pP.trsf.rz=l_nData[5]
         cls()
        return
      break


      case 277,255

        cls()
        return
      break

      case 270
        call Float_Edit(l_nData[l_nSelectIndex],nPanelLTopX+7,l_nSelectIndex+nPanelLTopY+1)
      break

    endSwitch

    if l_nKey!=-1
      l_sItem[0]="X    :"+toString(".3",l_nData[0])
      l_sItem[1]="y    :"+toString(".3",l_nData[1])
      l_sItem[2]="Z    :"+toString(".3",l_nData[2])
      l_sItem[3]="RX   :"+toString(".3",l_nData[3])
      l_sItem[4]="RY   :"+toString(".3",l_nData[4])
      l_sItem[5]="RZ   :"+toString(".3",l_nData[5])
      call Control_List(l_sItem,l_nSelectIndex)

    endIf






  endWhile





end

--- Control_Preset.pgx ---
public program Control_Preset(num& x_nPreset[] (dimensions=2), num x_nIndex)
  local string l_sItem[5]
  local num l_nNum
  local num l_nKey
  local num l_nData[5]
  local num l_nSelectIndex
begin

  //修改点位的 joint

  for l_nNum=0 to 4
    l_nData[l_nNum]=x_nPreset[x_nIndex,l_nNum]
  endFor



  l_sItem[0]="激光功率  :"+toString("",l_nData[0])
  l_sItem[1]="气体压力  :"+toString("",l_nData[1])
  l_sItem[2]="占空比频率:"+toString("",l_nData[2])
  l_sItem[3]="激光占空比:"+toString("",l_nData[3])
  l_sItem[4]="随动高度  :"+toString("",l_nData[4])

  call Control_BottomS(",,,,,,取消,确定")
  call Control_PanelXY(8,0,15,5)
  call Control_Panel("工艺值")
  call Control_List(l_sItem,l_nSelectIndex)
  while true
    l_nKey=getKey()

    switch l_nKey
      case 261
        l_nSelectIndex=max(0,l_nSelectIndex-1)
      break

      case 266
        l_nSelectIndex=min(l_nSelectIndex+1,5)
      break

      case 278
        for l_nNum=0 to 4
          x_nPreset[x_nIndex,l_nNum]=min(max(l_nData[l_nNum],0),100)
        endFor
        return
      break


      case 277
        return
      break

      case 270
        call Float_Edit(l_nData[l_nSelectIndex],nPanelLTopX+12,l_nSelectIndex+nPanelLTopY+1)
        l_nData[l_nSelectIndex]=min(max(l_nData[l_nSelectIndex],0),100)
      break

    endSwitch

    if l_nKey!=-1

      l_sItem[0]="激光功率  :"+toString("",l_nData[0])
      l_sItem[1]="气体压力  :"+toString("",l_nData[1])
      l_sItem[2]="占空比频率:"+toString("",l_nData[2])
      l_sItem[3]="激光占空比:"+toString("",l_nData[3])
      l_sItem[4]="随动高度  :"+toString("",l_nData[4])
      call Control_List(l_sItem,l_nSelectIndex)

    endIf






  endWhile





end

--- Control_Recipe.pgx ---
public program Control_Recipe(trsf& x_trFrame, trsf& x_trOffset)
  local num l_nSelectIndex
  local num l_nData[30]
  local num l_nKey
  local num l_nNum
begin
//产品的参数



  //主要是用户坐标系和偏移
  l_nData[0]=x_trFrame.x
  l_nData[1]=x_trFrame.y
  l_nData[2]=x_trFrame.z
  l_nData[3]=x_trFrame.rx
  l_nData[4]=x_trFrame.ry
  l_nData[5]=x_trFrame.rz

  l_nData[6]=x_trOffset.x
  l_nData[7]=x_trOffset.y
  l_nData[8]=x_trOffset.z
  l_nData[9]=x_trOffset.rx
  l_nData[10]=x_trOffset.ry
  l_nData[11]=x_trOffset.rz


  resize(sBuff,1,12)

  sBuff[0]="坐标系X  :"+toString(".3",l_nData[0])
  sBuff[1]="坐标系y  :"+toString(".3",l_nData[1])
  sBuff[2]="坐标系Z  :"+toString(".3",l_nData[2])
  sBuff[3]="坐标系RX :"+toString(".3",l_nData[3])
  sBuff[4]="坐标系RY :"+toString(".3",l_nData[4])
  sBuff[5]="坐标系RZ :"+toString(".3",l_nData[5])


  sBuff[6]="偏移 X   :"+toString(".3",l_nData[6])
  sBuff[7]="偏移 y   :"+toString(".3",l_nData[7])
  sBuff[8]="偏移 Z   :"+toString(".3",l_nData[8])
  sBuff[9]="偏移 RX  :"+toString(".3",l_nData[9])
  sBuff[10]="偏移 RY  :"+toString(".3",l_nData[10])
  sBuff[11]="偏移 RZ  :"+toString(".3",l_nData[11])





  call Control_BottomS(",,,,,,取消,确定")
  call Control_PanelXY(8,0,17,12)
  call Control_Panel("产品参数")
  call Control_List(sBuff,l_nSelectIndex)
  while true
    l_nKey=getKey()

    switch l_nKey
      case 261
        //        l_nSelectIndex=max(0,l_nSelectIndex-1)

        l_nSelectIndex=l_nSelectIndex-1
        if l_nSelectIndex<=-1
          l_nSelectIndex=size(sBuff)-1
        endIf

      break

      case 266
        l_nSelectIndex=l_nSelectIndex+1
        if l_nSelectIndex>=size(sBuff)
          l_nSelectIndex=0
        endIf
        //l_nSelectIndex=min(l_nSelectIndex+1,size(sBuff)-1)
      break

      case 278
        x_trFrame.x=l_nData[0]
        x_trFrame.y =l_nData[1]
        x_trFrame.z=l_nData[2]
        x_trFrame.rx =l_nData[3]
        x_trFrame.ry =l_nData[4]
        x_trFrame.rz =l_nData[5]

        x_trOffset.x=l_nData[6]
        x_trOffset.y =l_nData[7]
        x_trOffset.z =l_nData[8]
        x_trOffset.rx =l_nData[9]
        x_trOffset.ry =l_nData[10]
        x_trOffset.rz =l_nData[11]




        cls()
        return
      break


      case 277
        cls()
        return
      break

      case 270
        call Float_Edit(l_nData[l_nSelectIndex],nPanelLTopX+11,l_nSelectIndex+nPanelLTopY+1)

      break


    endSwitch

    if l_nKey!=-1

      sBuff[0]="坐标系X  :"+toString(".3",l_nData[0])
      sBuff[1]="坐标系y  :"+toString(".3",l_nData[1])
      sBuff[2]="坐标系Z  :"+toString(".3",l_nData[2])
      sBuff[3]="坐标系RX :"+toString(".3",l_nData[3])
      sBuff[4]="坐标系RY :"+toString(".3",l_nData[4])
      sBuff[5]="坐标系RZ :"+toString(".3",l_nData[5])


      sBuff[6]="偏移 X   :"+toString(".3",l_nData[6])
      sBuff[7]="偏移 y   :"+toString(".3",l_nData[7])
      sBuff[8]="偏移 Z   :"+toString(".3",l_nData[8])
      sBuff[9]="偏移 RX  :"+toString(".3",l_nData[9])
      sBuff[10]="偏移 RY  :"+toString(".3",l_nData[10])
      sBuff[11]="偏移 RZ  :"+toString(".3",l_nData[11])
      call Control_List(sBuff,l_nSelectIndex)

    endIf


  endWhile



end

--- Control_Remote.pgx ---
public program Control_Remote(num& x_nMode, num& x_nCycleCount)
  local string l_sItem[2]
  local num l_nNum
  local num l_nKey
  local num l_nData[2]
  local num l_nSelectIndex
  local string l_sSMess[6]
begin

  //修改点位的 joint
  l_nData[0]=max(round(x_nMode),0)
  l_nData[1]=max(round(x_nCycleCount),0)

  l_sSMess[0]="按钮触发单工位"
  l_sSMess[1]="按钮触发单周期"
  l_sSMess[2]="按钮触发多周期"
  l_sSMess[3]="无需按钮触发"
  l_sSMess[4]="按钮触发排队"
  l_sSMess[5]="用户自定义触发"


  l_sItem[0]="生产模式:"+l_sSMess[l_nData[0]]
  l_sItem[1]="周期次数:"+toString("",l_nData[1])


  call Control_BottomS(",,,,,,取消,确定")
  call Control_PanelXY(8,0,25,2)
  call Control_ListCls()
  call Control_Panel("生产配置")
  call Control_List(l_sItem,l_nSelectIndex)
  while true
    l_nKey=getKey()

    switch l_nKey
      case 261
        l_nSelectIndex=max(0,l_nSelectIndex-1)
      break

      case 266
        l_nSelectIndex=min(l_nSelectIndex+1,1)
      break

      case 278
        x_nMode=l_nData[0]
        x_nCycleCount=l_nData[1]

        return
      break


      case 277
        return
      break

      case 270
        if l_nSelectIndex==0
         call Sel_Edit(l_nData[0],nPanelLTopX+10,nPanelLTopY+1,l_sSMess)
        else
          call Float_Edit(l_nData[1],nPanelLTopX+10,nPanelLTopY+2)

        endIf



        l_nData[l_nSelectIndex]=max(round(l_nData[l_nSelectIndex]),0)
      break

    endSwitch

    if l_nKey!=-1
  l_sItem[0]="生产模式:"+l_sSMess[l_nData[0]]
  l_sItem[1]="周期次数:"+toString("",l_nData[1])
      call Control_List(l_sItem,l_nSelectIndex)

    endIf






  endWhile





end

--- Control_Scara.pgx ---
public program Control_Scara()
  local string l_sText[20]
  local num l_nIndex
begin
//   l_sText[0]="       .:i.         "
//   l_sText[1]="         .:i.       "
//   l_sText[2]="       Xzi  iU    , "
//   l_sText[3]="     .6:     .i   : "
//   l_sText[4]="    .A    MM .E:,.n."
//   l_sText[5]="    6     8MvYIZX;v."
//   l_sText[6]="   7.     vi;iCCviX "
//   l_sText[7]="   7 :.   vtYn7Yci7 "
//   l_sText[8]="    .7Co622onU  6t; "
//   l_sText[9]="  SY7Az      .  .:Q."
//   l_sText[10]="  MMMMM           X "
//   l_sText[11]="  MM:..    "
//   l_sText[12]="  MMt:;  "
//   l_sText[13]="  MMt:;  "




   l_sText[0]="         .--.           "
   l_sText[1]="      :./    \ ..   .     "
   l_sText[2]="    .:/    |::::.;:..:   "
   l_sText[3]="   ../     |::::;;:.:     "
   l_sText[4]="   ./ . ...:i:;..:::     "
   l_sText[5]="  . .i;.......  :.;      "
   l_sText[6]="   |::|           |:|             "
   l_sText[7]=" |::. .|              "
   l_sText[8]=" |::.  |               "
   l_sText[9]=" | .:::|                "
   l_sText[10]=" |  .ri|             "
   l_sText[11]=" |r72r7|            "
   l_sText[12]=" |scara|            "


for l_nIndex=0 to 9
  gotoxy(18,l_nIndex+1)
  put(left(l_sText[l_nIndex],22))
endFor
















end

--- Control_Traj.pgx ---
public program Control_Traj(trsf& x_trFrame, trsf& x_trOffset, trsf& x_trArray, trsf& x_trDownLead, trsf& x_trWorkPlace, bool& x_bInerCut, num& x_nDelay[], num& x_nLength[])
  local num l_nSelectIndex
  local num l_nData[31]
  local num l_nKey
  local num l_nNum
begin
  //修改点位的 joint


  // x_trDownLead.rz只能是大于10
  //圆弧度
  l_nData[10]=x_trFrame.x
  l_nData[11]=x_trFrame.y
  l_nData[12]=x_trFrame.z
  l_nData[13]=x_trFrame.rx
  l_nData[14]=x_trFrame.ry
  l_nData[15]=x_trFrame.rz

  l_nData[16]=x_trOffset.x
  l_nData[17]=x_trOffset.y
  l_nData[18]=x_trOffset.z
  l_nData[19]=x_trOffset.rx
  l_nData[20]=x_trOffset.ry
  l_nData[21]=x_trOffset.rz

  l_nData[2]=x_trArray.x
  l_nData[3]=x_trArray.y
  l_nData[4]=x_trArray.z
  l_nData[5]=x_trArray.rx

  l_nData[6]=x_trDownLead.x
  l_nData[7]=x_trDownLead.y
  l_nData[8]=x_trDownLead.z
  l_nData[9]=x_trDownLead.rx

  l_nData[0]=x_trDownLead.ry
  l_nData[1]=x_trDownLead.rz*10

  l_nData[22]=x_trWorkPlace.x
  l_nData[23]=x_trWorkPlace.y

  l_nData[24]=sel(x_bInerCut,0,1)
  l_nData[25]=x_nDelay[0]
  l_nData[26]=x_nDelay[1]
  l_nData[27]=x_nLength[0]
  l_nData[28]=x_nLength[1]
  l_nData[29]=x_trWorkPlace.ry
  l_nData[30]=x_trWorkPlace.rz
  resize(sData,1,3)
  sData[0]="无"
  sData[1]="直线"
  sData[2]="圆弧"

  resize(sBuff,1,31)
  sBuff[0]="圆直径   :"+toString(".3",l_nData[0])
  sBuff[1]="圆弧度   :"+toString(".3",l_nData[1])

  sBuff[2]="X方向个数:"+toString("",l_nData[2])
  sBuff[3]="X方向距离:"+toString(".3",l_nData[3])
  sBuff[4]="Y方向个数:"+toString("",l_nData[4])
  sBuff[5]="Y方向距离:"+toString(".3",l_nData[5])

  sBuff[6]="引入类型 :"+sData[l_nData[6]]
  sBuff[7]="引入比例 :"+toString(".3",l_nData[7])
  sBuff[8]="引出类型 :"+sData[l_nData[8]]
  sBuff[9]="引出比例 :"+toString(".3",l_nData[9])



  sBuff[10]="坐标系X  :"+toString(".3",l_nData[10])
  sBuff[11]="坐标系y  :"+toString(".3",l_nData[11])
  sBuff[12]="坐标系Z  :"+toString(".3",l_nData[12])
  sBuff[13]="坐标系RX :"+toString(".3",l_nData[13])
  sBuff[14]="坐标系RY :"+toString(".3",l_nData[14])
  sBuff[15]="坐标系RZ :"+toString(".3",l_nData[15])


  sBuff[16]="偏移 X   :"+toString(".3",l_nData[16])
  sBuff[17]="偏移 y   :"+toString(".3",l_nData[17])
  sBuff[18]="偏移 Z   :"+toString(".3",l_nData[18])
  sBuff[19]="偏移 RX  :"+toString(".3",l_nData[19])
  sBuff[20]="偏移 RY  :"+toString(".3",l_nData[20])
  sBuff[21]="偏移 RZ  :"+toString(".3",l_nData[21])


  sBuff[22]="七轴距离 :"+toString(".3",l_nData[22])
  sBuff[23]="七轴速度 :"+toString(".3",l_nData[23])
  sBuff[25]="激光开延时:"+toString(".3",l_nData[25])
  sBuff[26]="激光关延时:"+toString(".3",l_nData[26])
  sBuff[27]="边长1    :"+toString(".3",l_nData[27])
  sBuff[28]="边长2    :"+toString(".3",l_nData[28])
  sBuff[29]="收弧长度 :"+toString(".3",l_nData[29])
  resize(sData,1,2)
  sData[0]="内切"
  sData[1]="外切"
  sBuff[24]="类型     :"+sData[l_nData[24]]
  sBuff[30]="打孔工艺 :"+toString(".3",l_nData[30])


  call Control_BottomS(",,,,,,取消,确定")
  call Control_PanelXY(8,0,17,11)
  call Control_Panel("路径参数")
  call Control_List(sBuff,l_nSelectIndex)
  while true
    l_nKey=getKey()

    switch l_nKey
      case 261
        //        l_nSelectIndex=max(0,l_nSelectIndex-1)

        l_nSelectIndex=l_nSelectIndex-1
        if l_nSelectIndex<=-1
          l_nSelectIndex=size(sBuff)-1
        endIf

      break

      case 266
        l_nSelectIndex=l_nSelectIndex+1
        if l_nSelectIndex>=size(sBuff)
          l_nSelectIndex=0
        endIf
        //l_nSelectIndex=min(l_nSelectIndex+1,size(sBuff)-1)
      break

      case 278
        x_trFrame.x=l_nData[10]
        x_trFrame.y =l_nData[11]
        x_trFrame.z=l_nData[12]
        x_trFrame.rx =l_nData[13]
        x_trFrame.ry =l_nData[14]
        x_trFrame.rz =l_nData[15]

        x_trOffset.x=l_nData[16]
        x_trOffset.y =l_nData[17]
        x_trOffset.z =l_nData[18]
        x_trOffset.rx =l_nData[19]
        x_trOffset.ry =l_nData[20]
        x_trOffset.rz =l_nData[21]

        x_trArray.x=l_nData[2]
        x_trArray.y= l_nData[3]
        x_trArray.z= l_nData[4]
        x_trArray.rx= l_nData[5]

        x_trDownLead.x= l_nData[6]
        x_trDownLead.y= l_nData[7]
        x_trDownLead.z= l_nData[8]
        x_trDownLead.rx= l_nData[9]
        x_trDownLead.ry= l_nData[0]
        x_trDownLead.rz= l_nData[1]/10

        x_trWorkPlace.x= l_nData[22]
        x_trWorkPlace.y= l_nData[23]
        x_bInerCut=l_nData[24]==0
        x_nDelay[0]=l_nData[25]
        x_nDelay[1]=l_nData[26]
        x_nLength[0]=l_nData[27]
        x_nLength[1]=l_nData[28]
        x_trWorkPlace.ry=l_nData[29]
        x_trWorkPlace.rz=min(50,max(l_nData[30],1))
        cls()
        return
      break


      case 277,255
        cls()
        return
      break

      case 270
        switch l_nSelectIndex
          case 4,30
            call Int_Edit(l_nData[l_nSelectIndex],nPanelLTopX+11,sel(l_nSelectIndex>=10,10,l_nSelectIndex)+nPanelLTopY+1)
          break

          case 0,1,2,3,5,7,9,10,11,12,13,14,15,16,17,18,19,20,21,22,23,25,26,27,28,29
            call Float_Edit(l_nData[l_nSelectIndex],nPanelLTopX+11,sel(l_nSelectIndex>=10,10,l_nSelectIndex)+nPanelLTopY+1)
          break
          case 6,8,24
            if l_nSelectIndex>9
              resize(sData,1,2)
              sData[0]="内切"
              sData[1]="外切"
            else
              resize(sData,1,3)
              sData[0]="无"
              sData[1]="直线"
              sData[2]="圆弧"
            endIf
            call Sel_Edit(l_nData[l_nSelectIndex],nPanelLTopX+11,sel(l_nSelectIndex>=10,10,l_nSelectIndex)+nPanelLTopY+1,sData)

          break


        endSwitch
      break


    endSwitch

    if l_nKey!=-1

      resize(sData,1,3)
      sData[0]="无"
      sData[1]="直线"
      sData[2]="圆弧"

      resize(sBuff,1,31)
      sBuff[0]="圆直径   :"+toString(".3",l_nData[0])
      sBuff[1]="圆弧度   :"+toString(".3",l_nData[1])

      sBuff[2]="X方向个数:"+toString("",l_nData[2])
      sBuff[3]="X方向距离:"+toString(".3",l_nData[3])
      sBuff[4]="Y方向个数:"+toString("",l_nData[4])
      sBuff[5]="Y方向距离:"+toString(".3",l_nData[5])

      sBuff[6]="引入类型 :"+sData[l_nData[6]]
      sBuff[7]="引入比例 :"+toString(".3",l_nData[7])
      sBuff[8]="引出类型 :"+sData[l_nData[8]]
      sBuff[9]="引出比例 :"+toString(".3",l_nData[9])



      sBuff[10]="坐标系X  :"+toString(".3",l_nData[10])
      sBuff[11]="坐标系y  :"+toString(".3",l_nData[11])
      sBuff[12]="坐标系Z  :"+toString(".3",l_nData[12])
      sBuff[13]="坐标系RX :"+toString(".3",l_nData[13])
      sBuff[14]="坐标系RY :"+toString(".3",l_nData[14])
      sBuff[15]="坐标系RZ :"+toString(".3",l_nData[15])


      sBuff[16]="偏移 X   :"+toString(".3",l_nData[16])
      sBuff[17]="偏移 y   :"+toString(".3",l_nData[17])
      sBuff[18]="偏移 Z   :"+toString(".3",l_nData[18])
      sBuff[19]="偏移 RX  :"+toString(".3",l_nData[19])
      sBuff[20]="偏移 RY  :"+toString(".3",l_nData[20])
      sBuff[21]="偏移 RZ  :"+toString(".3",l_nData[21])


      sBuff[22]="七轴距离 :"+toString(".3",l_nData[22])
      sBuff[23]="七轴速度 :"+toString(".3",l_nData[23])
      resize(sData,1,2)
      sData[0]="内切"
      sData[1]="外切"
      sBuff[24]="类型     :"+sData[l_nData[24]]
      sBuff[25]="激光开延时:"+toString(".3",l_nData[25])
      sBuff[26]="激光关延时:"+toString(".3",l_nData[26])
      sBuff[27]="边长1    :"+toString(".3",l_nData[27])
      sBuff[28]="边长2    :"+toString(".3",l_nData[28])
      sBuff[29]="收弧长度 :"+toString(".3",l_nData[29])
      sBuff[30]="打孔工艺 :"+toString(".3",l_nData[30])
      call Control_List(sBuff,l_nSelectIndex)

    endIf






  endWhile









end

--- Control_YesNO.pgx ---
public program Control_YesNO(string x_sTitle, bool& x_bRes)
begin



  x_bRes=false
  call Control_PanelMd(x_sTitle)
  call Control_BottomS(",,,,,,是,否")

  while true
    switch getKey()

      //F8
      case 278
        x_bRes=false
        cls()
        return
      break
      //F7
      case  277
         x_bRes=true
         cls()
        return
      break
    endSwitch
    delay(0)
  endWhile
end

--- Form_4jHome.pgx ---
public program Form_4jHome(string x_sTitle, jointRs& x_jJ)
begin
  //call Form_MainS(",,,,,记录,保存,退出")
  title(x_sTitle)

  call Form_PattenS(x_sTitle,"记录,,,,,,保存,退出","记录,,,,,,保存,退出")
  call Control_PanelXY(22,0,15,10)
  call Control_Panel("Home")
  //call con
  gotoxy(nPanelLTopX+1,nPanelLTopY+1)
  put(left("j1:"+toString(".3",x_jJ.j1)+"        ",nPanelWidthX))

  gotoxy(nPanelLTopX+1,nPanelLTopY+2)
  put(left("j2:"+toString(".3",x_jJ.j2)+"        ",nPanelWidthX))

  gotoxy(nPanelLTopX+1,nPanelLTopY+3)
  put(left("j3:"+toString(".3",x_jJ.j3)+"        ",nPanelWidthX))

  gotoxy(nPanelLTopX+1,nPanelLTopY+4)
  put(left("j4:"+toString(".3",x_jJ.j4)+"        ",nPanelWidthX))



end

--- Form_Action.pgx ---
public program Form_Action(string x_sTitle, string x_sPanelTitle, string& x_sList[], num& x_nSelectIndex, bool& x_bIO[], num x_nPresetIndex, string& x_sLable[])
  local num l_nNum
begin

 // cls()
  x_nSelectIndex=round(x_nSelectIndex)%500
  x_nPresetIndex=x_nPresetIndex%50
  title(x_sTitle)
   gotoxy(0,0)
  put("动作执行需上电!")
  gotoxy(0,2)
  put("动作参数:")





  call Control_PanelXY(22,0,15,10)
    for l_nNum=0 to size(x_sLable)-1
    gotoxy(0,l_nNum+3)
    put(left(x_sLable[l_nNum]+"                            ",nPanelLTopX-1))
    endFor
  call Control_Panel(x_sPanelTitle)
  setTextMode(sel(x_bIO[0],1,0))
  gotoxy(1,13)
  put("执行")

 setTextMode(0)

        gotoxy(21,13)
    put("上传")
    gotoxy(31,13)
    put("保存")

    gotoxy(26,13)
    put("修改")
    gotoxy(31,13)
    put("保存")

    gotoxy(36,13)
    put("退出")


  call Control_List(x_sList,x_nSelectIndex)



end

--- FORM_BYE.pgx ---
public program Form_Bye()
begin
 cls()
 call Control_PanelMd("感谢使用史陶比尔机器人软件")



end

--- Form_Config.pgx ---
public program Form_Config(num& x_nNum[], num& x_nPointIndex)
  local string l_sBuff[2]
  local string l_sVersion
begin



  l_sBuff[0]="关"
  l_sBuff[1]="开"
  //轮询
  resize(sBuff,1,40)

  sBuff[0]="工具(Tool)X  :"+toString(".3",  x_nNum[0])
  sBuff[1]="工具(Tool)Y  :"+toString(".3",x_nNum[1])
  sBuff[2]="工具(Tool)Z  :"+toString(".3",x_nNum[2])
  sBuff[3]="工具(Tool)RX :"+toString(".3",x_nNum[3])
  sBuff[4]="工具(Tool)RY :"+toString(".3",x_nNum[4])
  sBuff[5]="工具(Tool)RZ :"+toString(".3",x_nNum[5])


  sBuff[6]="回零速度(m/min):"+toString(".3",x_nNum[6])
  sBuff[7]="不拆工具示教 :"+l_sBuff[x_nNum[7]]
  sBuff[8]="示教回退(启动:"+l_sBuff[x_nNum[8]]

  sBuff[9]="PWM频率高(HZ):"+toString(".3",x_nNum[9])
  sBuff[10]="PWM频率低(HZ):"+toString(".3",x_nNum[10])
  sBuff[11]="模拟量系数   :"+toString(".3",x_nNum[11])
  sBuff[12]="速度匹配(s)  :"+toString(".3",x_nNum[12])
  sBuff[13]="光斑补偿(mm) :"+toString(".3",x_nNum[13])


  sBuff[14]="开气延时(s)  :"+toString(".3",x_nNum[14])
  sBuff[15]="随动延时(s)  :"+toString(".3",x_nNum[15])
  sBuff[16]="工位延时(s)  :"+toString(".3",x_nNum[16])

  sBuff[17]="快捷速度(mm/s):"+toString("",x_nNum[17])
  sBuff[18]="快捷加速度(%):"+toString("",x_nNum[18])
  sBuff[19]="快捷Blend(mm):"+toString(".3",x_nNum[19])
  sBuff[20]="快捷工艺     :"+toString("",x_nNum[20])


  sBuff[21]="异步7轴(启动):"+l_sBuff[x_nNum[21]]
  sBuff[22]="7轴home点(mm):"+toString(".3",x_nNum[22])
  sBuff[23]="7轴分度      :"+toString(".3",x_nNum[23])
  sBuff[24]="7轴安全点速度:"+toString("",x_nNum[24])



  sBuff[25]="焊接(启动)   :"+l_sBuff[x_nNum[25]]
  sBuff[26]="焊接回退长度 :"+toString("",x_nNum[26])
  //sBuff[27]="步进(启动)   :"+l_sBuff[x_nNum[27]]
  sBuff[28]="步进距离(mm) :"+toString(".3",x_nNum[28])
  sBuff[29]="远程生产密码 :"+toString(".3",x_nNum[29])
  sBuff[30]="同工位多产品 :"+l_sBuff[x_nNum[30]]
  sBuff[27]="报警延时触发 :"+toString(".3",x_nNum[27])
  sBuff[31]="拐角速度自适 :"+l_sBuff[x_nNum[31]]


  sBuff[32]="异步8轴(启动):"+l_sBuff[x_nNum[32]]
  sBuff[33]="8轴home点(mm):"+toString(".3",x_nNum[33])
  sBuff[34]="8轴分度      :"+toString(".3",x_nNum[34])
  sBuff[35]="8轴安全点速度:"+toString("",x_nNum[35])



  call Control_LeftS(",,,,,上传,保存,退出,")
  call Control_PanelS("选项",17,0,20,10)
  call Control_BottomS(",,,,,上传,保存,退出,")
  call Control_List(sBuff,x_nPointIndex)







end

--- Form_Main.pgx ---
public program Form_Main(string& x_sBottomList[])
  local num l_nIndex
begin
  //欢迎界面，显示日期和时间
 userPage()
cls()
 call Control_PanelMd("机器人处在空闲界面")



//     for l_nIndex=0 to min(7,size(x_sBottomList)-1)
//    gotoxy(1+l_nIndex*5,13)
//    if size(x_sBottomList)>l_nIndex and x_sBottomList[l_nIndex]!=""
//      put(x_sBottomList[l_nIndex])
//    endIf
//    endFor
 call Control_Bottom(x_sBottomList)
end

--- Form_MainS.pgx ---
public program Form_MainS(string x_sBottomList)
  local num l_nIndex
  local bool l_bRes
  local string l_sBuff[20]
begin
  //把字符串给分开，使用,作为分隔符
  call Str_SplitComma(l_bRes,x_sBottomList,l_sBuff)
  if !l_bRes
    return
  endIf
   call Form_Main(l_sBuff)
end

--- Form_Product.pgx ---
public program Form_Product(string x_sTitle, string& x_sLableList[], string& x_sList[], string x_sBottom)
  local num l_nNum
begin

//cls()
title(x_sTitle)
setTextMode(0)
for l_nNum=0 to size(x_sLableList)-1
  gotoxy(0,l_nNum+1)

  put(left(x_sLableList[l_nNum]+"            ",18))
  gotoxy(22,l_nNum+1)

   put(left(x_sList[l_nNum]+"            ",18))
endFor

call Control_BottomS(x_sBottom)



end

--- Form_ScaraRobot.pgx ---
public program Form_ScaraRobot()
begin
 call Form_PattenS("Scara1.0:主界面","示教Home,示教TCP,示教码垛,产品编辑,,选项,高级,退出","F1,F2,F3,F4,F5,F6,F7,F8")
 call Control_Scara()

end

--- Form_SelSharp.pgx ---
public program Form_SelSharp(num& x_nTypeIndex, bool& x_bRes)
  local string l_sList[12]
  local num l_nKey
  local num l_nIndex
begin
  l_nIndex=0
  l_sList[0]="不规则图形"
  l_sList[1]="圆-圆心直径法"
  l_sList[2]="圆-三点法"
  l_sList[3]="三角形"
  l_sList[4]="矩形"
  l_sList[5]="正五边形"
  l_sList[6]="正六边形"
  l_sList[7]="腰形"
  l_sList[8]="五角星"
  l_sList[9]="圆管"
  l_sList[10]="C形-三点法"


  cls()
  //title(x_sTitle)

  call Control_PanelXY(0,0,15,10)
  call Control_Panel("图形类型")
  call Control_BottomS("示教,,,,,,,退出")

  //x_nSelectIndex=0
  call Control_List(l_sList,l_nIndex)

  while true
    l_nKey=getKey()
    switch l_nKey
      case 261
        l_nIndex=max(l_nIndex-1,0)
      break

      case 266
        l_nIndex=min(l_nIndex+1,10)
      break

      //示教,F1 和回车键
      case 271,270
        x_bRes=true
        switch l_nIndex
          case 0
            x_nTypeIndex=10
          break

          case 1
            x_nTypeIndex=2
          break

          case 2
            x_nTypeIndex=1
          break

          case 3
            x_nTypeIndex=3
          break

          case 4
            x_nTypeIndex=4
          break

          case 5
            x_nTypeIndex=5
          break

          case 6
            x_nTypeIndex=6
          break


          case 7
            x_nTypeIndex=7
          break



          case 8
            x_nTypeIndex=21
          break


          case 9
            x_nTypeIndex=22
          break


          case 10
            x_nTypeIndex=24
          break
        endSwitch

        return
      break

      //F8 和ESC键退出
      case 278,255
        x_bRes=false
        return

      break



    endSwitch

    if l_nKey!=-1

      call Control_List(l_sList,l_nIndex)
    endIf


  endWhile




end

--- Form_Simulation.pgx ---
public program Form_Simulation(string x_sTitle, string x_sPanelTitle, string& x_sList[], num& x_nSelectIndex, num& x_nPreset[], bool& x_bIO[])
begin

  //cls()
  x_nSelectIndex=round(x_nSelectIndex)%500

  title(x_sTitle)
  gotoxy(1,4)
  put("实时工艺参数:")


  if x_sPanelTitle=="切割点" or x_sPanelTitle=="工艺表"
    gotoxy(1,5)
    put("激光功率  :"+toString("",x_nPreset[0])+"   ")
    gotoxy(1,6)
    put("气体压力  :"+toString("",x_nPreset[3])+"   ")
    gotoxy(1,7)
    put("占空比频率:"+toString("",x_nPreset[1])+"   ")
    gotoxy(1,8)
    put("激光占空比:"+toString("",x_nPreset[2])+"   ")
    gotoxy(1,9)
    put("随动高度  :"+toString("",x_nPreset[4])+"   ")
  else
    gotoxy(1,5)
    put("激光功率  :0   ")
    gotoxy(1,6)
    put("气体压力  :0   ")
    gotoxy(1,7)
    put("占空比频率:0   ")
    gotoxy(1,8)
    put("激光占空比:0   ")
    gotoxy(1,9)
    put("随动高度  :0   ")

  endIf


  call Control_PanelXY(22,0,15,10)
  call Control_Panel(x_sPanelTitle)
  //call Control_BottomS("激光,随动,气体,,,,,终止")
  setTextMode(sel(x_bIO[0],1,0))
  gotoxy(1,13)
  put("激光")


  setTextMode(sel(x_bIO[1],1,0))
  gotoxy(6,13)
  put("随动")


  setTextMode(sel(x_bIO[2],01,0))
  gotoxy(11,13)
  put("气体")

  setTextMode(0)

  if  x_sPanelTitle=="工艺表"

    gotoxy(21,13)
    put("上传")

    gotoxy(26,13)
    put("修改")
    gotoxy(31,13)
    put("保存")

    gotoxy(36,13)
    put("退出")

  else
    gotoxy(36,13)
    put("终止")

  endIf
  //x_nSelectIndex=0
  call Control_List(x_sList,x_nSelectIndex)



end

--- INT_EDIT.pgx ---
program Int_Edit(num& x_nData, num x_nX, num x_nY)
  local num l_nKey
  local num l_nNum
begin

  call Int_EditS(x_nData,x_nX,x_nY,"")
end

--- SEL_EDIT.pgx ---
public program Sel_Edit(num& x_nData, num x_nX, num x_nY, string& x_sMess[])
  local num l_nKey
  local num l_nNum
  local num l_nBuff
begin
  //说明
  //函数功能：上下进行选择
  //x_nData 被选中的字符串数组序号
  //x_sMess  可选字符串数组
  //x_nX x_nY 被选中的起始点




  //参数判断
  x_nX=min(max(0,x_nX),39)
  x_nY=min(max(0,x_nY),nPanelLTopY+nPanelLengthY)
  x_nData=max(min(x_nData,size(x_sMess)-1),0)

  l_nNum=x_nData
  l_nKey=0
  l_nBuff=l_nNum-100


  //按键选择
  while l_nKey!=270 and l_nKey!=255

    //对按键进行判断
    l_nKey=getKey()
    switch l_nKey
      //向下
      case 261
        l_nNum=min(l_nNum-1,0)
        if l_nNum<=-1
          l_nNum=size(x_sMess)-1
        endIf
      break

      //向上
      case 266
        l_nNum=l_nNum+1
        if l_nNum>=size(x_sMess)
          l_nNum=0
        endIf
      break
      //回车
      case 270
        x_nData=l_nNum
        return
      break
    endSwitch

    //重新刷新界面
    if l_nBuff!=l_nNum
      l_nBuff=l_nNum
      gotoxy(x_nX,x_nY)
      setTextMode(0)
      put(left(x_sMess[l_nNum]+"           ",nPanelWidthX-x_nX+nPanelLTopX))
    endIf


  endWhile
end

--- STR_EDIT.pgx ---
program Str_Edit(string& x_sData, num x_nX, num x_nY)
  local string l_sBuff
  local num l_nKey
  local string l_sOri
begin

  x_nX=min(max(0,x_nX),39)
  x_nY=min(max(0,x_nY),13)
 // x_nLength=min(max(0,x_nLength),39)
  l_sOri=x_sData

  setTextMode(1)
  l_nKey=0
  l_sBuff=x_sData
  while l_nKey!=270 and l_nKey!=255
    gotoxy(x_nX,x_nY)
    setTextMode(0)
    put(left("                              ",nPanelWidthX-x_nX+nPanelLTopX))
    gotoxy(x_nX,x_nY)
    setTextMode(1)
    l_nKey=get(l_sBuff)
    //Enter
    if l_nKey==270
      setTextMode(0)
      x_sData=l_sBuff
    endIf
    //ESC
    if l_nKey==255
      setTextMode(0)
      x_sData= l_sOri
      setTextMode(0)
    endIf
    gotoxy(x_nX,x_nY)
    put(left(l_sBuff+"                    ",nPanelWidthX-x_nX+nPanelLTopX))
    delay(0)
  endWhile
end
